// TIA Portal V19 export
TYPE "LEXCHANGETRAY_typeVfdContronNode"
// commandConfiguration: LBC_typeSinaSpeedCommandConfiguration
// commands: LBC_typeSinaSpeedControlNodeCommands
// monitoring: LEXCHANGETRAY_typeVfdContronNodeMonitoring
// stored: Access Published
   STRUCT
      commandConfiguration : "LBC_typeSinaSpeedCommandConfiguration";
      commands : "LBC_typeSinaSpeedControlNodeCommands";
      monitoring { S7_SetPoint := 'True'} : "LEXCHANGETRAY_typeVfdContronNodeMonitoring";
   END_STRUCT;
END_TYPE
